(* Logix 5000 project; controller cal1615 1756-L62 rev 20.11; software revision 20.05; part 67 of 82 *)
(* tags used below, declared in another part *)
   FAULT : BOOL;   // Fault AFI
   p01_recipe_active : recipe;   // Active Recipe
   p01r02 : routine;   // System Misc Control
   p01r09_pb_global_reset : BOOL;   // System Modes PB: Global Fault Reset
   p02_dint_from_hmi : hmi_dint;
   p27_ao_dia_a : REAL;   // Lower Poly Letoff Analog Input Letoff A Diameter
   p27_ao_dia_b : REAL;   // Lower Poly Letoff Analog Input Letoff B Diameter
   p27_inactive_tension_sp : REAL;   // Lower Poly Letoff Tension Inactive Tension Setpoint
   p27r01 : routine;   // Winder Main
   p27r03_lower_A_tension_on : BOOL;
   p27r03_lower_B_tension_on : BOOL;
   p27r05_lla_mode_tension : BOOL;   // Lower Poly Letoff Modes A Tension Mode
   p27r05_llb_mode_tension : BOOL;   // Lower Poly Letoff Modes B Tension Mode
   p27r09 : routine;   // Winder Modes
   p27r09_a_enable_toggle : SYS_Toggle;   // Lower Poly Letoff Modes A Toggle
   p27r09_b_enable_toggle : SYS_Toggle;   // Lower Poly Letoff Modes B Toggle
   p27r09_timer_fault : TIMER[4];   // Winder Modes Fault Delay
   p27r09_timer_warning : TIMER[4];   // Winder Modes Warning Delay
   p27r10 : routine;   // Winder Winder Speed
   p27r10_lla_selected_tension : REAL;   // Lower Poly Letoff Tension A Selected Tension
   p27r10_llb_selected_tension : REAL;   // Lower Poly Letoff Tension B Selected Tension
   p27r10_timer_fault : TIMER[4];   // Winder Fault Delay
   p27r10_timer_warning : TIMER[4];   // Winder Warning Delay
   p27r10_unwind_a_brake_torque : REAL;   // Lower Poly Letoff Tension Letoff A Brake Torque [lb-ft]
   p27r10_unwind_a_dia_ft : REAL;   // Lower Poly Letoff Tension Diameter A [ft]
   p27r10_unwind_b_brake_torque : REAL;   // Lower Poly Letoff Tension Letoff B Brake Torque [lb-ft]
   p27r10_unwind_b_dia_ft : REAL;   // Lower Poly Letoff Tension Diameter B [ft]
   p28_ai_slitter_amps : REAL;
   p28_ai_slitter_hz : REAL;
   p28_ai_slitter_speed : REAL;
   p28_di_brake : BOOL;
   p28_di_motor : BOOL;
   p28_di_slitter : acs800_di_normal;
   p28_dint_to_hmi : DINT[16];
   p28_do_slt_air_supply_sv : BOOL;
   p28r01 : routine;
   p28r02 : routine;
   p28r02_fault_exists : BOOL;
   p28r02_timer_fault : TIMER[4];
   p28r02_timer_warning : TIMER[4];
   p28r02_unack_fault : BOOL;
   p28r02_unack_warning : BOOL;
   p28r02_warning_exists : BOOL;
   p28r03 : routine;
   p28r03_hz : SYS_SCP;
   p28r03_slitter_speed_fb : SYS_RPM_TO_SPEED;
   p28r03_timer_fault : TIMER[4];
   p28r03_timer_warning : TIMER[4];
   p28r04 : routine;
   p28r04_slitter_gear_ratio : REAL;
   p28r04_slitter_roll_diameter_ft : REAL;
   p28r05 : routine;
   p28r06 : routine;
   p28r07 : routine;
   p28r08 : routine;
   p28r09 : routine;
   p28r11 : routine;
   p28r11_slitter_on : BOOL;
(* P27_Lower_Poly_Letoff, continued *)

ROUTINE R09_Modes   (* ladder *)
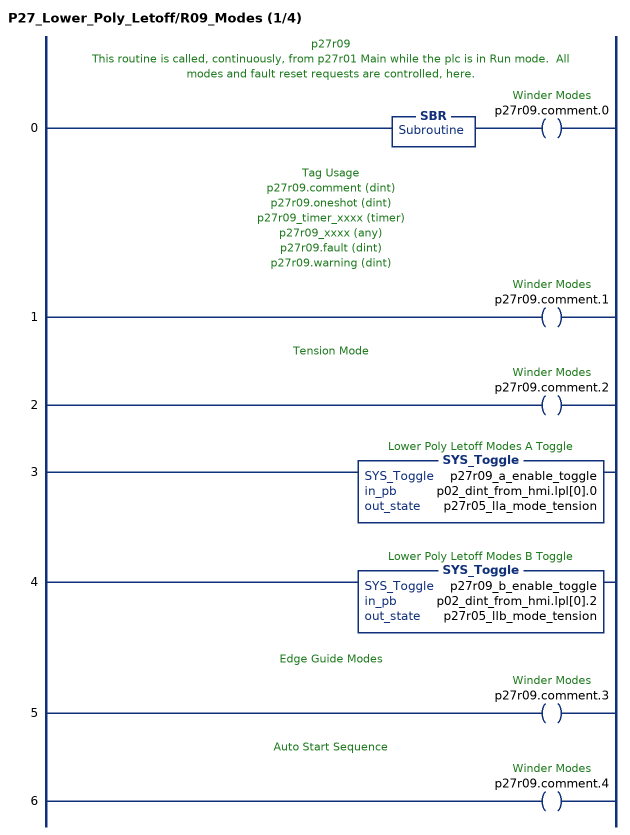
   // p27r09
   // This routine is called, continuously, from p27r01 Main while the plc is in Run mode.  All modes and fault reset requests are controlled, here.
   0: SBR()OTE(p27r09.comment.0);
   // Tag Usage
   // p27r09.comment (dint)
   // p27r09.oneshot (dint)
   // p27r09_timer_xxxx (timer)
   // p27r09_xxxx (any)
   // p27r09.fault (dint)
   // p27r09.warning (dint)
   1: OTE(p27r09.comment.1);
   // Tension Mode
   2: OTE(p27r09.comment.2);
   3: SYS_Toggle(p27r09_a_enable_toggle,p02_dint_from_hmi.lpl[0].0,p27r05_lla_mode_tension);
   4: SYS_Toggle(p27r09_b_enable_toggle,p02_dint_from_hmi.lpl[0].2,p27r05_llb_mode_tension);
   // Edge Guide Modes
   5: OTE(p27r09.comment.3);
   // Auto Start Sequence
   6: OTE(p27r09.comment.4);
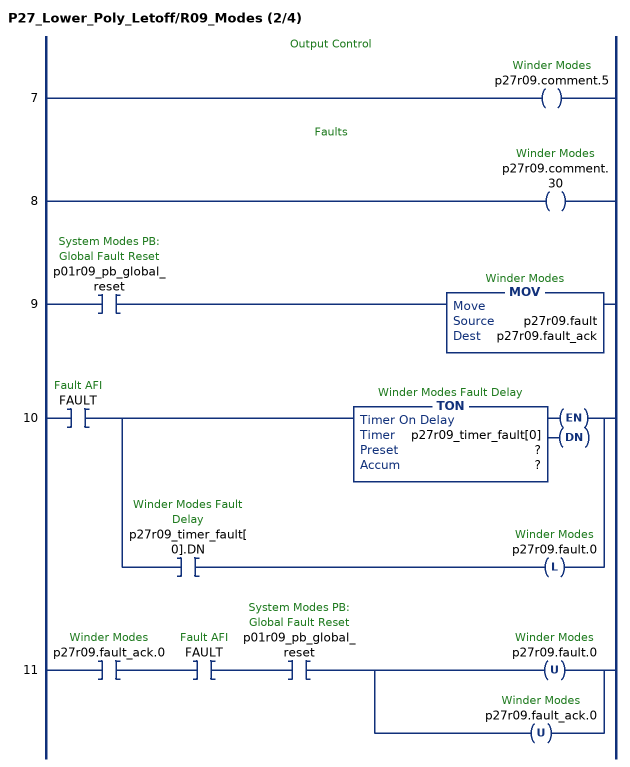
   // Output Control
   7: OTE(p27r09.comment.5);
   // Faults
   8: OTE(p27r09.comment.30);
   9: XIC(p01r09_pb_global_reset)MOV(p27r09.fault,p27r09.fault_ack);
   10: XIC(FAULT)[TON(p27r09_timer_fault[0],?,?) ,XIC(p27r09_timer_fault[0].DN) OTL(p27r09.fault.0) ];
   11: XIC(p27r09.fault_ack.0)XIC(FAULT)XIC(p01r09_pb_global_reset)[OTU(p27r09.fault.0) ,OTU(p27r09.fault_ack.0) ];
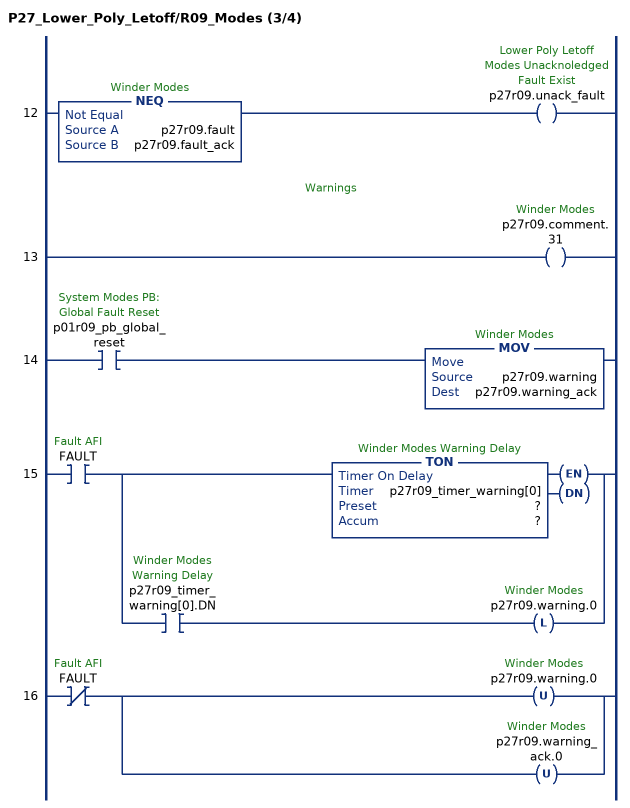
   12: NEQ(p27r09.fault,p27r09.fault_ack)OTE(p27r09.unack_fault);
   // Warnings
   13: OTE(p27r09.comment.31);
   14: XIC(p01r09_pb_global_reset)MOV(p27r09.warning,p27r09.warning_ack);
   15: XIC(FAULT)[TON(p27r09_timer_warning[0],?,?) ,XIC(p27r09_timer_warning[0].DN) OTL(p27r09.warning.0) ];
   16: XIO(FAULT)[OTU(p27r09.warning.0) ,OTU(p27r09.warning_ack.0) ];
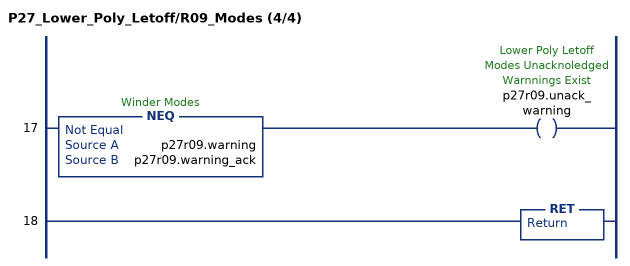
   17: NEQ(p27r09.warning,p27r09.warning_ack)OTE(p27r09.unack_warning);
   18: RET();
END_ROUTINE

ROUTINE R10_Tension   (* ladder *)
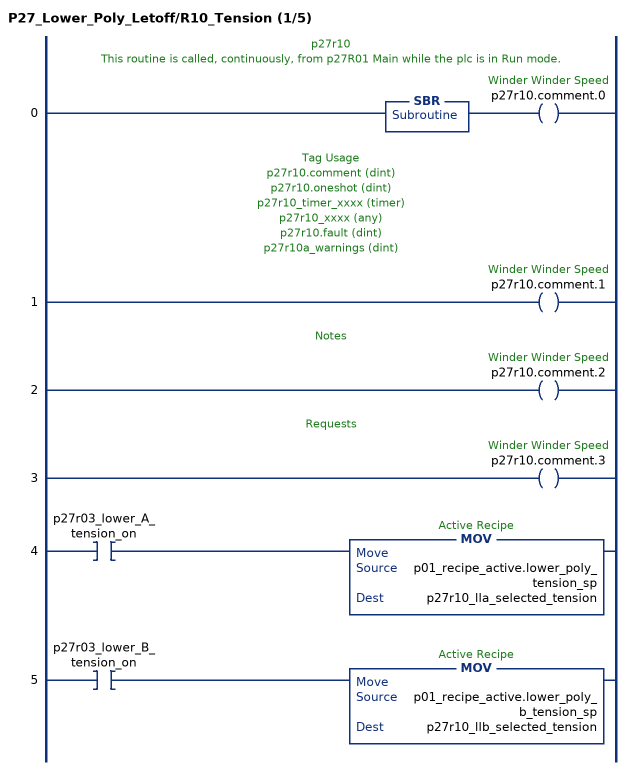
   // p27r10
   // This routine is called, continuously, from p27R01 Main while the plc is in Run mode.
   0: SBR()OTE(p27r10.comment.0);
   // Tag Usage
   // p27r10.comment (dint)
   // p27r10.oneshot (dint)
   // p27r10_timer_xxxx (timer)
   // p27r10_xxxx (any)
   // p27r10.fault (dint)
   // p27r10a_warnings (dint)
   1: OTE(p27r10.comment.1);
   // Notes
   2: OTE(p27r10.comment.2);
   // Requests
   3: OTE(p27r10.comment.3);
   4: XIC(p27r03_lower_A_tension_on)MOV(p01_recipe_active.lower_poly_tension_sp,p27r10_lla_selected_tension);
   5: XIC(p27r03_lower_B_tension_on)MOV(p01_recipe_active.lower_poly_b_tension_sp,p27r10_llb_selected_tension);
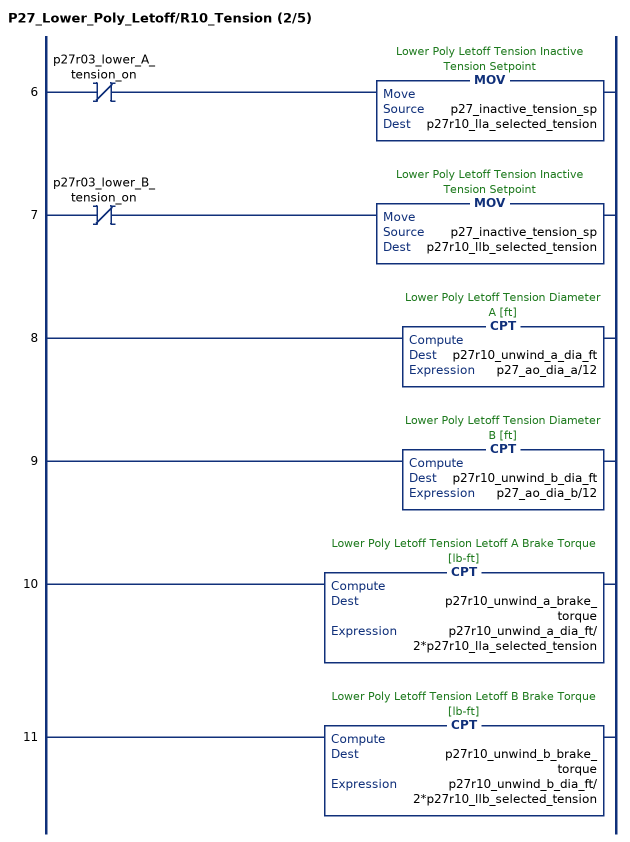
   6: XIO(p27r03_lower_A_tension_on)MOV(p27_inactive_tension_sp,p27r10_lla_selected_tension);
   7: XIO(p27r03_lower_B_tension_on)MOV(p27_inactive_tension_sp,p27r10_llb_selected_tension);
   8: CPT(p27r10_unwind_a_dia_ft,p27_ao_dia_a/12);
   9: CPT(p27r10_unwind_b_dia_ft,p27_ao_dia_b/12);
   10: CPT(p27r10_unwind_a_brake_torque,p27r10_unwind_a_dia_ft/2*p27r10_lla_selected_tension);
   11: CPT(p27r10_unwind_b_brake_torque,p27r10_unwind_b_dia_ft/2*p27r10_llb_selected_tension);
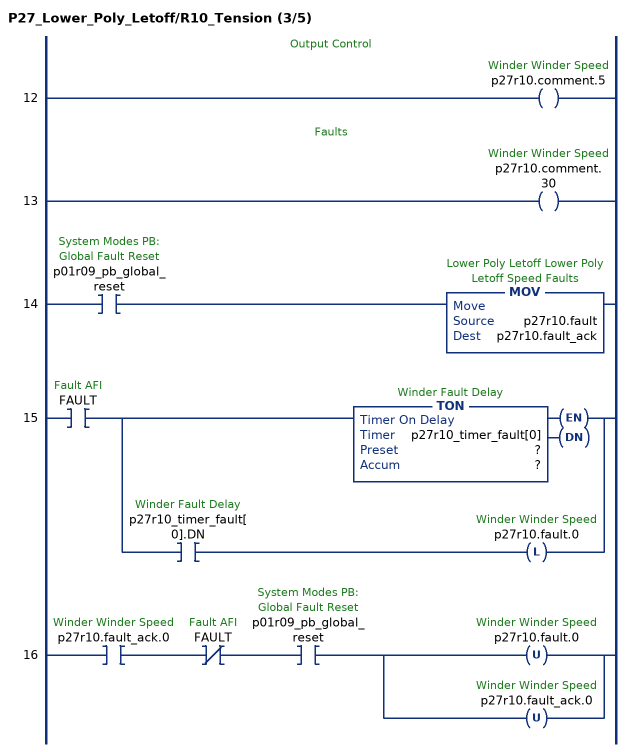
   // Output Control
   12: OTE(p27r10.comment.5);
   // Faults
   13: OTE(p27r10.comment.30);
   14: XIC(p01r09_pb_global_reset)MOV(p27r10.fault,p27r10.fault_ack);
   15: XIC(FAULT)[TON(p27r10_timer_fault[0],?,?) ,XIC(p27r10_timer_fault[0].DN) OTL(p27r10.fault.0) ];
   16: XIC(p27r10.fault_ack.0)XIO(FAULT)XIC(p01r09_pb_global_reset)[OTU(p27r10.fault.0) ,OTU(p27r10.fault_ack.0) ];
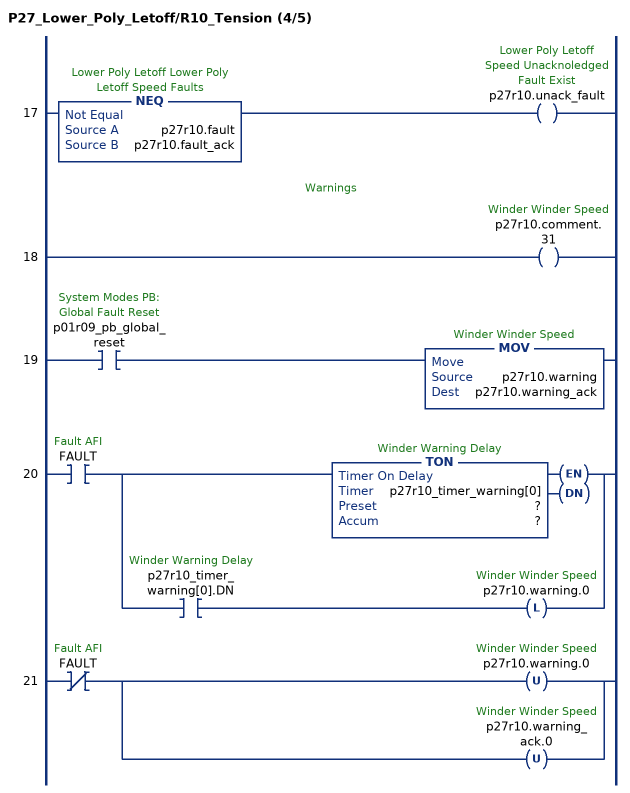
   17: NEQ(p27r10.fault,p27r10.fault_ack)OTE(p27r10.unack_fault);
   // Warnings
   18: OTE(p27r10.comment.31);
   19: XIC(p01r09_pb_global_reset)MOV(p27r10.warning,p27r10.warning_ack);
   20: XIC(FAULT)[TON(p27r10_timer_warning[0],?,?) ,XIC(p27r10_timer_warning[0].DN) OTL(p27r10.warning.0) ];
   21: XIO(FAULT)[OTU(p27r10.warning.0) ,OTU(p27r10.warning_ack.0) ];
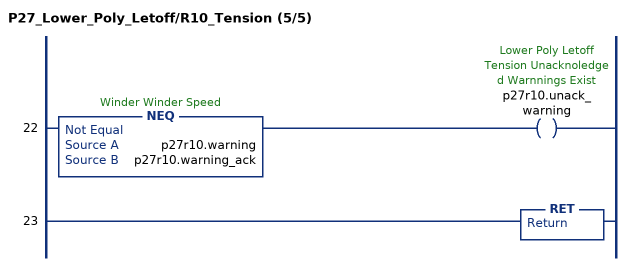
   22: NEQ(p27r10.warning,p27r10.warning_ack)OTE(p27r10.unack_warning);
   23: RET();
END_ROUTINE
END_PROGRAM

PROGRAM P28_Slitter   (* main routine R01_Main *)

ROUTINE R01_Main   (* ladder *)
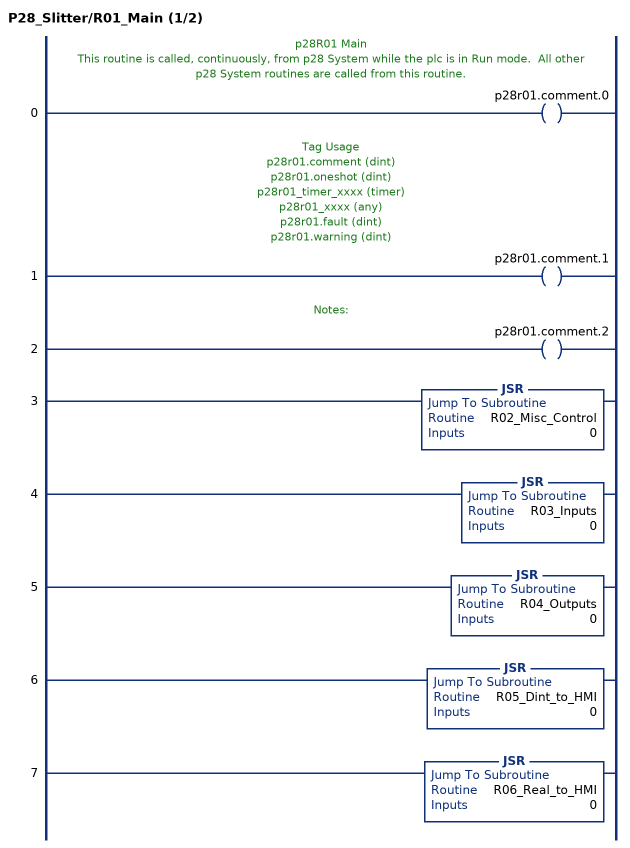
   // p28R01 Main
   // This routine is called, continuously, from p28 System while the plc is in Run mode.  All other p28 System routines are called from this routine.
   0: OTE(p28r01.comment.0);
   // Tag Usage
   // p28r01.comment (dint)
   // p28r01.oneshot (dint)
   // p28r01_timer_xxxx (timer)
   // p28r01_xxxx (any)
   // p28r01.fault (dint)
   // p28r01.warning (dint)
   1: OTE(p28r01.comment.1);
   // Notes:
   2: OTE(p28r01.comment.2);
   3: JSR(R02_Misc_Control,0);
   4: JSR(R03_Inputs,0);
   5: JSR(R04_Outputs,0);
   6: JSR(R05_Dint_to_HMI,0);
   7: JSR(R06_Real_to_HMI,0);
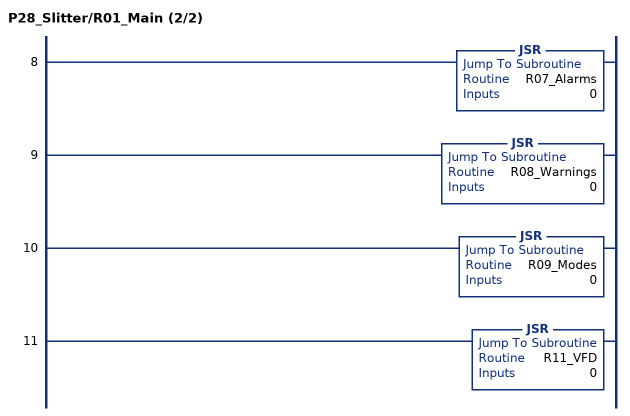
   8: JSR(R07_Alarms,0);
   9: JSR(R08_Warnings,0);
   10: JSR(R09_Modes,0);
   11: JSR(R11_VFD,0);
END_ROUTINE

ROUTINE R02_Misc_Control   (* ladder *)
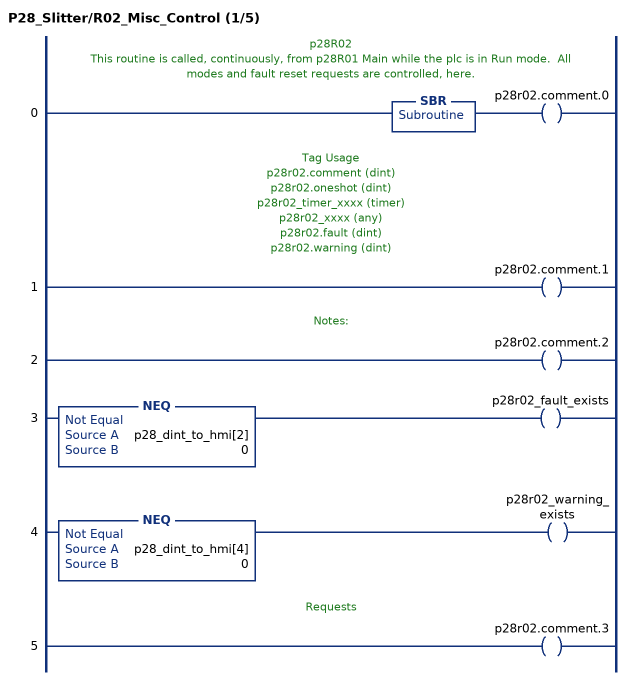
   // p28R02
   // This routine is called, continuously, from p28R01 Main while the plc is in Run mode.  All modes and fault reset requests are controlled, here.
   0: SBR()OTE(p28r02.comment.0);
   // Tag Usage
   // p28r02.comment (dint)
   // p28r02.oneshot (dint)
   // p28r02_timer_xxxx (timer)
   // p28r02_xxxx (any)
   // p28r02.fault (dint)
   // p28r02.warning (dint)
   1: OTE(p28r02.comment.1);
   // Notes:
   2: OTE(p28r02.comment.2);
   3: NEQ(p28_dint_to_hmi[2],0)OTE(p28r02_fault_exists);
   4: NEQ(p28_dint_to_hmi[4],0)OTE(p28r02_warning_exists);
   // Requests
   5: OTE(p28r02.comment.3);
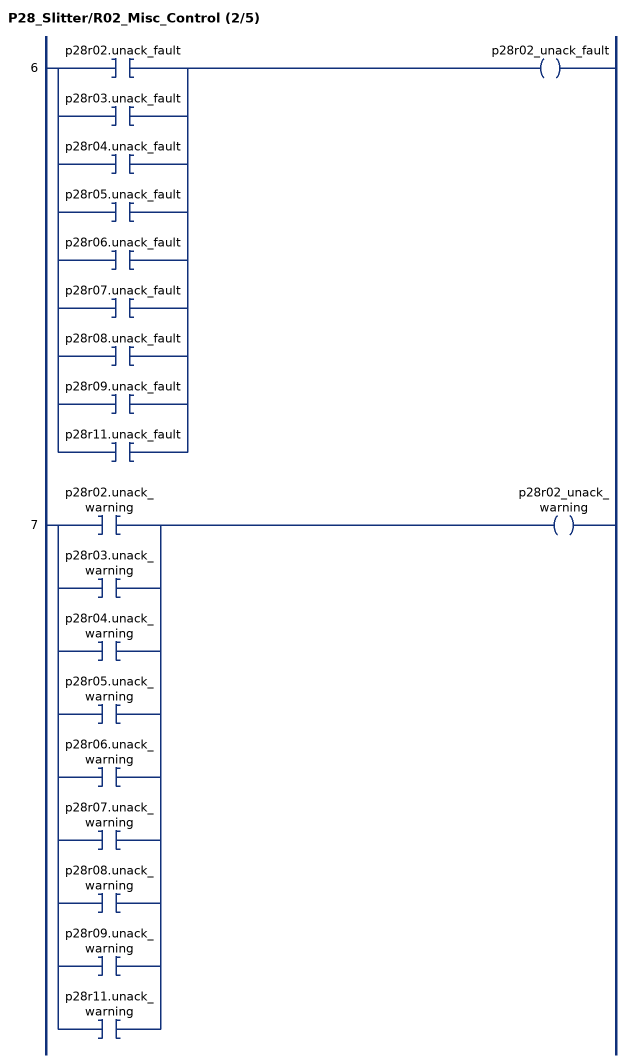
   6: [XIC(p28r02.unack_fault) ,XIC(p28r03.unack_fault) ,XIC(p28r04.unack_fault) ,XIC(p28r05.unack_fault) ,XIC(p28r06.unack_fault) ,XIC(p28r07.unack_fault) ,XIC(p28r08.unack_fault) ,XIC(p28r09.unack_fault) ,XIC(p28r11.unack_fault) ]OTE(p28r02_unack_fault);
   7: [XIC(p28r02.unack_warning) ,XIC(p28r03.unack_warning) ,XIC(p28r04.unack_warning) ,XIC(p28r05.unack_warning) ,XIC(p28r06.unack_warning) ,XIC(p28r07.unack_warning) ,XIC(p28r08.unack_warning) ,XIC(p28r09.unack_warning) ,XIC(p28r11.unack_warning) ]OTE(p28r02_unack_warning);
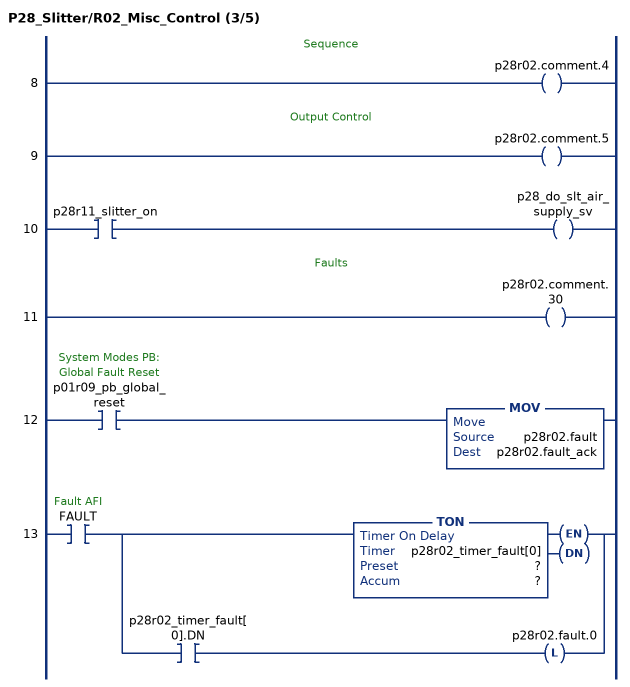
   // Sequence
   8: OTE(p28r02.comment.4);
   // Output Control
   9: OTE(p28r02.comment.5);
   10: XIC(p28r11_slitter_on)OTE(p28_do_slt_air_supply_sv);
   // Faults
   11: OTE(p28r02.comment.30);
   12: XIC(p01r09_pb_global_reset)MOV(p28r02.fault,p28r02.fault_ack);
   13: XIC(FAULT)[TON(p28r02_timer_fault[0],?,?) ,XIC(p28r02_timer_fault[0].DN) OTL(p28r02.fault.0) ];
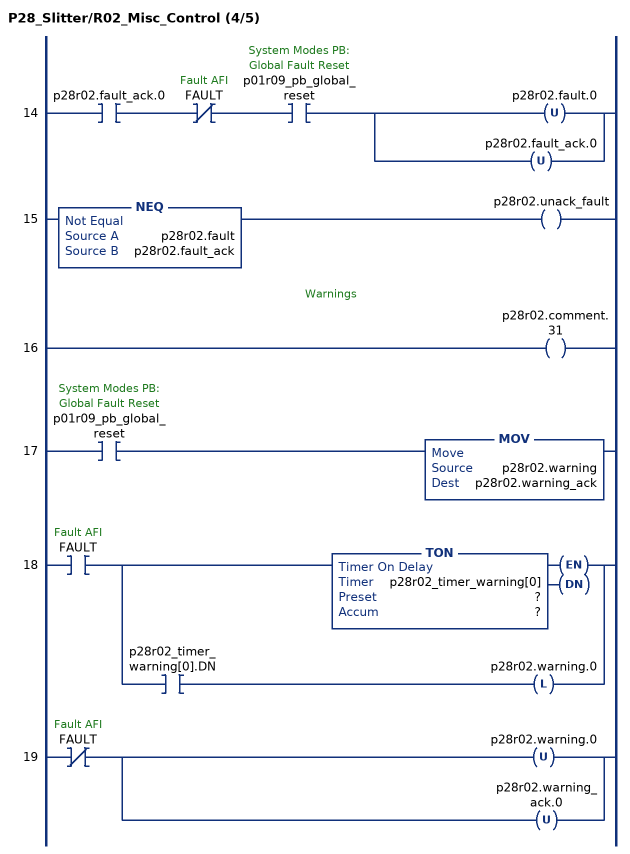
   14: XIC(p28r02.fault_ack.0)XIO(FAULT)XIC(p01r09_pb_global_reset)[OTU(p28r02.fault.0) ,OTU(p28r02.fault_ack.0) ];
   15: NEQ(p28r02.fault,p28r02.fault_ack)OTE(p28r02.unack_fault);
   // Warnings
   16: OTE(p28r02.comment.31);
   17: XIC(p01r09_pb_global_reset)MOV(p28r02.warning,p28r02.warning_ack);
   18: XIC(FAULT)[TON(p28r02_timer_warning[0],?,?) ,XIC(p28r02_timer_warning[0].DN) OTL(p28r02.warning.0) ];
   19: XIO(FAULT)[OTU(p28r02.warning.0) ,OTU(p28r02.warning_ack.0) ];
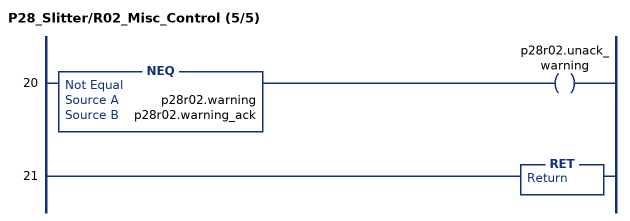
   20: NEQ(p28r02.warning,p28r02.warning_ack)OTE(p28r02.unack_warning);
   21: RET();
END_ROUTINE

ROUTINE R03_Inputs   (* ladder *)
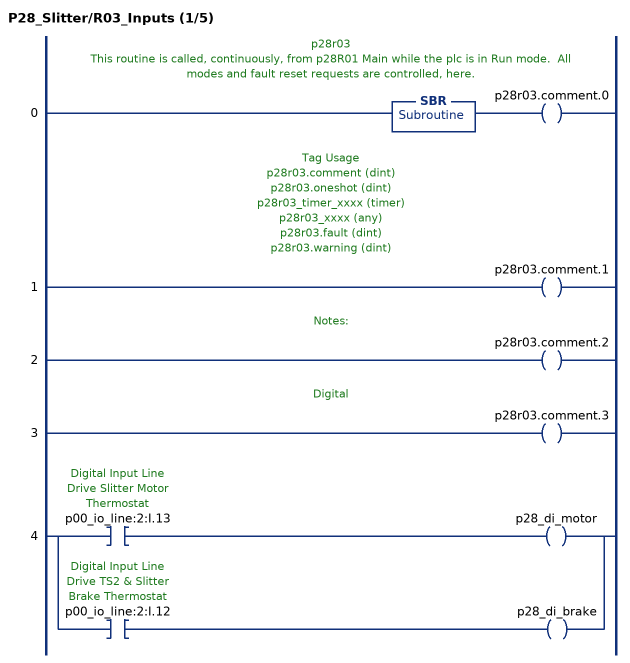
   // p28r03
   // This routine is called, continuously, from p28R01 Main while the plc is in Run mode.  All modes and fault reset requests are controlled, here.
   0: SBR()OTE(p28r03.comment.0);
   // Tag Usage
   // p28r03.comment (dint)
   // p28r03.oneshot (dint)
   // p28r03_timer_xxxx (timer)
   // p28r03_xxxx (any)
   // p28r03.fault (dint)
   // p28r03.warning (dint)
   1: OTE(p28r03.comment.1);
   // Notes:
   2: OTE(p28r03.comment.2);
   // Digital
   3: OTE(p28r03.comment.3);
   4: [XIC(p00_io_line:2:I.13) OTE(p28_di_motor) ,XIC(p00_io_line:2:I.12) OTE(p28_di_brake) ];
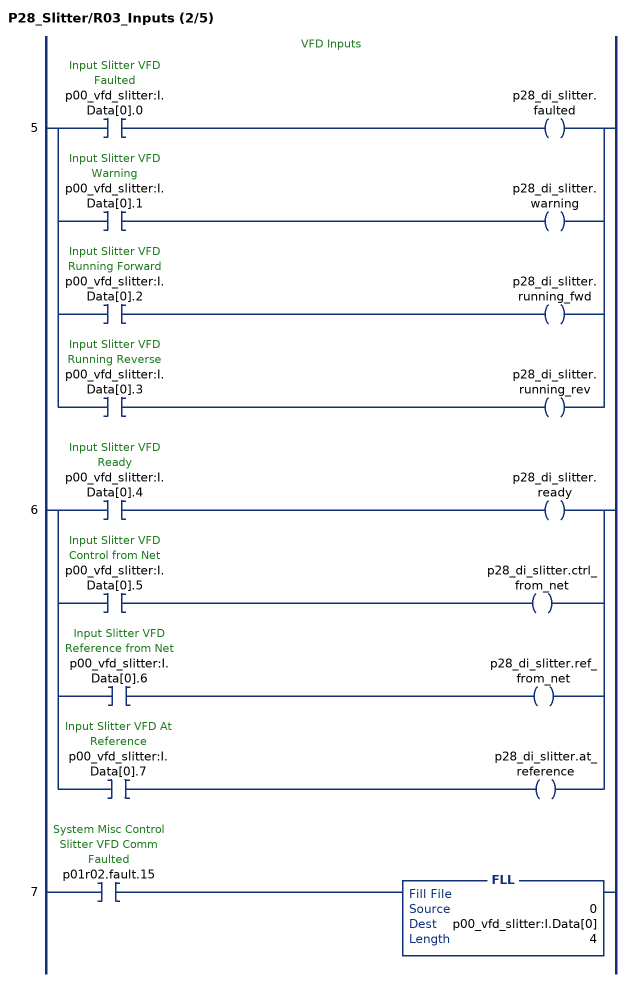
   // VFD Inputs
   5: [XIC(p00_vfd_slitter:I.Data[0].0) OTE(p28_di_slitter.faulted) ,XIC(p00_vfd_slitter:I.Data[0].1) OTE(p28_di_slitter.warning) ,XIC(p00_vfd_slitter:I.Data[0].2) OTE(p28_di_slitter.running_fwd) ,XIC(p00_vfd_slitter:I.Data[0].3) OTE(p28_di_slitter.running_rev) ];
   6: [XIC(p00_vfd_slitter:I.Data[0].4) OTE(p28_di_slitter.ready) ,XIC(p00_vfd_slitter:I.Data[0].5) OTE(p28_di_slitter.ctrl_from_net) ,XIC(p00_vfd_slitter:I.Data[0].6) OTE(p28_di_slitter.ref_from_net) ,XIC(p00_vfd_slitter:I.Data[0].7) OTE(p28_di_slitter.at_reference) ];
   7: XIC(p01r02.fault.15)FLL(0,p00_vfd_slitter:I.Data[0],4);
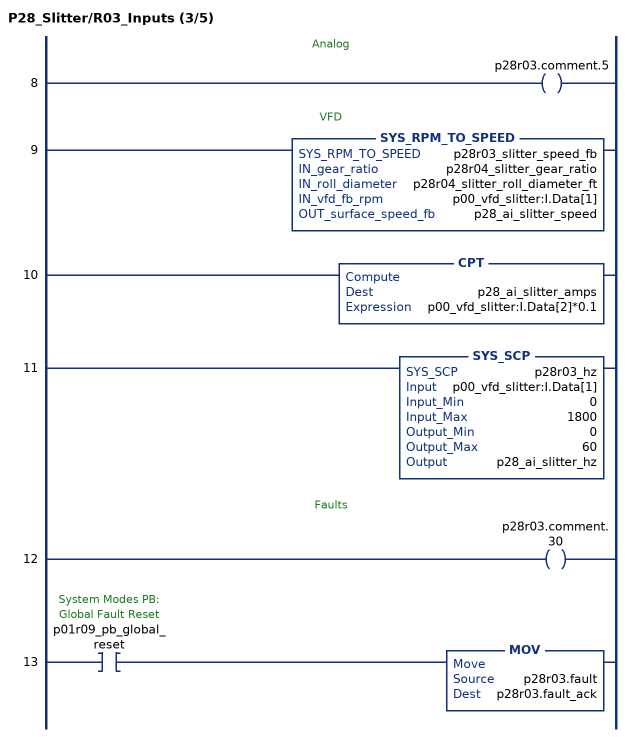
   // Analog
   8: OTE(p28r03.comment.5);
   // VFD
   9: SYS_RPM_TO_SPEED(p28r03_slitter_speed_fb,p28r04_slitter_gear_ratio,p28r04_slitter_roll_diameter_ft,p00_vfd_slitter:I.Data[1],p28_ai_slitter_speed);
   10: CPT(p28_ai_slitter_amps,p00_vfd_slitter:I.Data[2]*0.1);
   11: SYS_SCP(p28r03_hz,p00_vfd_slitter:I.Data[1],0,1800,0,60,p28_ai_slitter_hz);
   // Faults
   12: OTE(p28r03.comment.30);
   13: XIC(p01r09_pb_global_reset)MOV(p28r03.fault,p28r03.fault_ack);
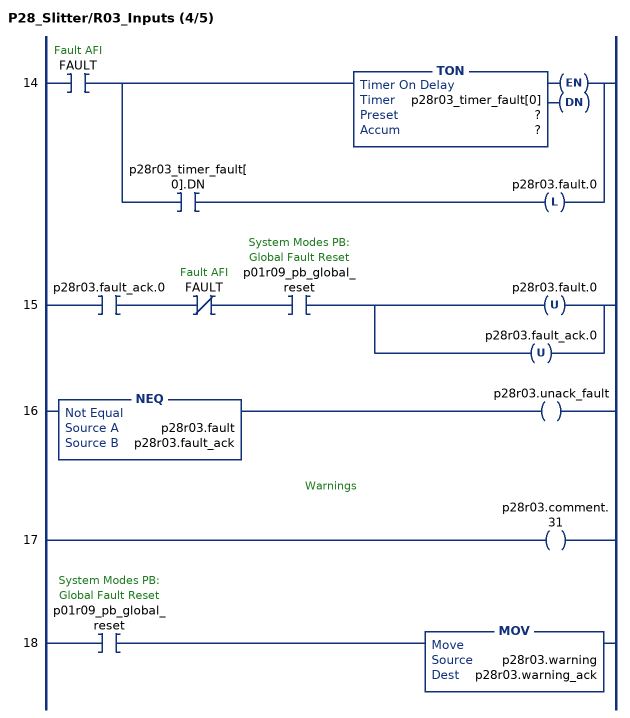
   14: XIC(FAULT)[TON(p28r03_timer_fault[0],?,?) ,XIC(p28r03_timer_fault[0].DN) OTL(p28r03.fault.0) ];
   15: XIC(p28r03.fault_ack.0)XIO(FAULT)XIC(p01r09_pb_global_reset)[OTU(p28r03.fault.0) ,OTU(p28r03.fault_ack.0) ];
   16: NEQ(p28r03.fault,p28r03.fault_ack)OTE(p28r03.unack_fault);
   // Warnings
   17: OTE(p28r03.comment.31);
   18: XIC(p01r09_pb_global_reset)MOV(p28r03.warning,p28r03.warning_ack);
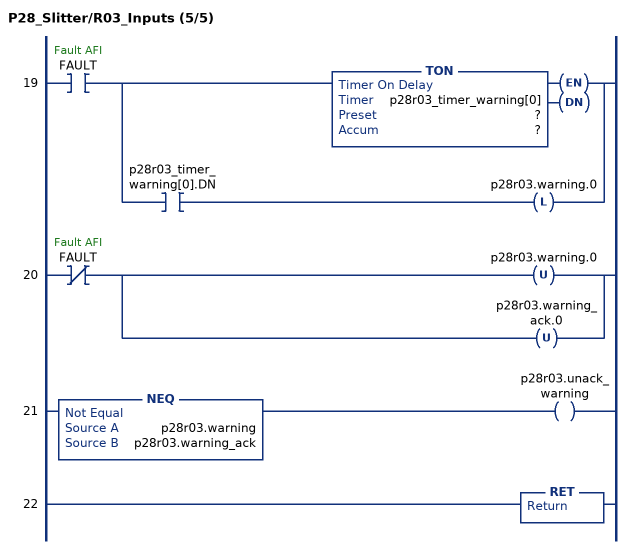
   19: XIC(FAULT)[TON(p28r03_timer_warning[0],?,?) ,XIC(p28r03_timer_warning[0].DN) OTL(p28r03.warning.0) ];
   20: XIO(FAULT)[OTU(p28r03.warning.0) ,OTU(p28r03.warning_ack.0) ];
   21: NEQ(p28r03.warning,p28r03.warning_ack)OTE(p28r03.unack_warning);
   22: RET();
END_ROUTINE
